// TIA Portal V18 export
DATA_BLOCK "PLC8_910A4_8DI_8DO_DO_Vars"   // DB11072
{ S7_Optimized_Access := 'FALSE' }
VERSION : 0.1
// stored: AutoNumber false, DBAccessibleFromOPCUA true, IsOnlyStoredInLoadMemory false, IsWriteProtectedInAS false
   VAR
      DO1 { S7_SetPoint := 'True'} : "UDT_DOadv";   // AHU F Дозвіл на роботу 1- ст. ККБ
      DO2 { S7_SetPoint := 'True'} : "UDT_DOadv";   // AHU F Дозвіл на роботу 2- ст. ККБ
      DO3 { S7_SetPoint := 'True'} : "UDT_DOadv";   // AHU F Дозвіл на роботу 3- ст. ККБ
      DO4 { S7_SetPoint := 'True'} : "UDT_DOadv";   // AHU F Дозвіл на роботу 4- ст. ККБ
      DO5 { S7_SetPoint := 'True'} : "UDT_DOadv";   // Резерв
      DO6 { S7_SetPoint := 'True'} : "UDT_DOadv";   // Резерв
      DO7 { S7_SetPoint := 'True'} : "UDT_DOadv";   // Резерв
      DO8 { S7_SetPoint := 'True'} : "UDT_DOadv";   // Резерв
   END_VAR
BEGIN
   DO1.iFuncSystemID := 10;
   DO1.iFuncVar := 10;
   DO2.iFuncSystemID := 10;
   DO2.iFuncVar := 11;
   DO3.iFuncSystemID := 10;
   DO3.iFuncVar := 12;
   DO4.iFuncSystemID := 100;
   DO4.iFuncVar := 1;
   DO5.iFuncSystemID := 100;
   DO5.iFuncVar := 5;
   DO6.iFuncSystemID := 100;
   DO6.iFuncVar := 3;
   DO7.iFuncSystemID := 10;
   DO7.iFuncVar := 5;
   DO8.iFuncSystemID := 10;
   DO8.iFuncVar := 6;
END_DATA_BLOCK
